TYPE ST_MotionRequest :
STRUCT
    bNewMoveReq: BOOL;
    nCmdData: INT;
    nCommand: INT;
    bExecute : BOOL;
    bExecHome: BOOL;
    bExecMove: BOOL;
    bStop : BOOL;
    bReset : BOOL;
    bEnable : BOOL;
    bPrepareDisable : BOOL;
END_STRUCT
END_TYPE

(* stored: Version 1.1.0.1
   DUT ST_MotionRequest: Id {a07ca9a6-ee49-49b8-ab2e-03bd2d0e53c7} *)
